{attribute 'GeneratedUsingTerminal: EL3423-0000-0020'}
{attribute addProperty BoxType "EL3423-0000-0020"}
{attribute addProperty Id "Reactive_EnergyAT %I*LINT8"}
{attribute addProperty CRC "545183756"}
{attribute addProperty Size "8"}
TYPE Total_Reactive_Reduced_207ED80C EXTENDS InputBase_8311D824 :
STRUCT
	{attribute addProperty Name "Reactive_Energy"}
	Reactive_Energy AT %I* : LINT;
END_STRUCT
END_TYPE

(* stored: Version 1.2.0.0, ProductVersion 3.1.4024.9
   DUT Total_Reactive_Reduced_207ED80C: Id {4ad0f863-5c2c-4302-8fdf-ddc073871ddc} *)
